{attribute addProperty BoxType "EL2596-0000-0017"}
{attribute addProperty Id "DOX_StatusAT %I*DOX_Status_95DEE7BC1620DOX_ControlAT %Q*DOX_Control_3320C5611620WcStateAT %I*WcState_F855686C1620InfoDataAT %I*InfoData_BC63D37F80100"}
{attribute addProperty CRC "274677248"}
{attribute addProperty SizeInBites "128"}
{attribute addProperty SizeInBytes "16"}
TYPE EL2596_AF8FAE89 :
STRUCT
	{attribute addProperty Name "DOX_Status"}
	DOX_Status : DOX_Status_95DEE7BC;
	{attribute addProperty Name "DOX_Control"}
	DOX_Control : DOX_Control_3320C561;
	{attribute addProperty Name "WcState"}
	WcState : WcState_F855686C;
	{attribute addProperty Name "InfoData"}
	InfoData : InfoData_BC63D37F;
END_STRUCT
END_TYPE

(* stored: Version 1.2.0.0, ProductVersion 3.1.4024.9
   DUT EL2596_AF8FAE89: Id {2fc4a8f3-bd0c-4f32-ae39-b9e8e69c3ed8} *)
